FUNCTION BYTE_TO_BOOLS
  (* Standard: 61499-1 *)
  (* Version 1.0, 2024-02-22, franz *)
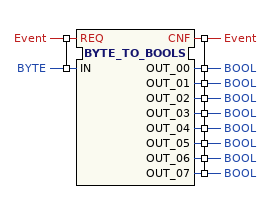
  EVENT_INPUT
    REQ WITH IN; (* Normal Execution Request *)
  END_EVENT
  EVENT_OUTPUT
    CNF WITH OUT_00, OUT_01, OUT_02, OUT_03, OUT_04, OUT_05, OUT_06, OUT_07; (* Execution Confirmation *)
  END_EVENT
  VAR_INPUT
    IN : BYTE; (* BYTE Input *)
  END_VAR
  VAR_OUTPUT
    OUT_00 : BOOL; (* BIT 00 *)
    OUT_01 : BOOL; (* BIT 01 *)
    OUT_02 : BOOL; (* BIT 02 *)
    OUT_03 : BOOL; (* BIT 03 *)
    OUT_04 : BOOL; (* BIT 04 *)
    OUT_05 : BOOL; (* BIT 05 *)
    OUT_06 : BOOL; (* BIT 06 *)
    OUT_07 : BOOL; (* BIT 07 *)
  END_VAR
  BODY IN ST:
FUNCTION BYTE_TO_BOOLS

VAR_INPUT
	IN : BYTE;    // BYTE Input
END_VAR

VAR_OUTPUT
	OUT_00 : BOOL;    // BIT 00
	OUT_01 : BOOL;    // BIT 01
	OUT_02 : BOOL;    // BIT 02
	OUT_03 : BOOL;    // BIT 03
	OUT_04 : BOOL;    // BIT 04
	OUT_05 : BOOL;    // BIT 05
	OUT_06 : BOOL;    // BIT 06
	OUT_07 : BOOL;    // BIT 07
END_VAR

(* this Function extracts the 8 BOOLS from a byte *)
OUT_00 := IN.0;
OUT_01 := IN.1;
OUT_02 := IN.2;
OUT_03 := IN.3;
OUT_04 := IN.4;
OUT_05 := IN.5;
OUT_06 := IN.6;
OUT_07 := IN.7;

END_FUNCTION
  END_BODY
END_FUNCTION
